ADAPTER AE (* unidirectional Adapter Interface for 1 Event *)
  (* Standard: 61499-1; Description: Copyright (c) 2025 HR Agrartechnik GmbH This program and the accompanying materials are made available under the terms of the Eclipse Public License 2.0 which is available at https://www.eclipse.org/legal/epl-2.0/ SPDX-License-Identifier: EPL-2.0 *)
  (* Version 1.0, 2025-01-24, Franz Höpfinger, HR Agrartechnik GmbH, Initial Version *)
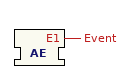
  EVENT_OUTPUT
    E1; (* Indication (or Request) *)
  END_EVENT
END_ADAPTER
